Fanuc KAREL source: FORCE_LINK.kl

PROGRAM T
%NOLOCKGROUP
VAR
 v0 : INTEGER
 v1 : STRING[40]
BEGIN
 FORCE_LINK(v0, v1)
END T
